FUNCTION_BLOCK FB_MoveZ_Exte
VAR_INPUT
	ref		:AXIS_REF;
	jogF	:BOOL;
	jogB	:BOOL;
	PosLimit			:BOOL;			(*正极限位信号*)
	NegLimit			:BOOL;			(*负极限位信号*)
	electromagnetLimit	:BOOL;
	
	maxDistance			:LREAL;			(*最大行程*)
	Acceleration		:LREAL;
	Deceleration		:LREAL;
	Jerk				:LREAL;
END_VAR
VAR_OUTPUT	
	electromagnet_power :BOOL;
END_VAR
VAR
	MC_Read:MC_ReadStatus;
	MC_ABS:MC_MoveAbsolute;
	MC_REL:MC_MoveRelative;
	MC_Jog:MC_Jog;	
	MC_VELO:MC_MoveVelocity;
	MC_stop:MC_Stop;
	
	step1,step2,step3		:INT;	
	R_TRIG1,R_TRIG2,R_TRIG3	:R_TRIG;
	R_TRIG_done				:R_TRIG;
	ton_NotMoving			:TON;
	ton_Moving				:TON;
	rel_do					:BOOL;
	abs_do					:BOOL;
	jogF_do					:BOOL;
	jogB_do					:BOOL;
	
	velo_do					:BOOL;
	stop_do					:BOOL;
	error					:BOOL;

	MoveAbsolute_Busy		:BOOL;
	MoveVelocity_Busy		:BOOL;
	MoveRelative_Busy		:BOOL;
	jog_EN					:BOOL;
	FB_START_r_trig:		R_TRIG;
	start					:BOOL;
	jog_f_trig				:F_TRIG;
END_VAR
VAR_IN_OUT 
	MoveRelExe					:BOOL;
	MoveAbsExe					:BOOL;
	MoveVelocityExe				:BOOL;//
	Velo						:LREAL;	//mm/s
	TargetRel					:LREAL;//mm
	TargetAbs					:LREAL;//mm
							
	Done						:BOOL;
	NotMovingTimeOut 			:BOOL;
	
END_VAR

(*********************NOT MOVING TIMEOUT***************************)
FB_START_r_trig(CLK:=jogF OR jogB OR MoveRelExe OR MoveAbsExe OR MoveVelocityExe  , Q=> );
IF FB_START_r_trig.Q THEN 
	start:=TRUE;
END_IF
ton_NotMoving(IN:=Ref.Status.NotMoving AND start  , PT:= T#5S, Q=> , ET=> );

Call_FB();
JOG();
MoveAbsolute();
MoveVelocity();
MoveRelative();


(*********************error***************************)
IF ton_NotMoving.Q OR error  THEN	
	start:=FALSE;
	NotMovingTimeOut:=TRUE;	
	error:=FALSE;
	ton_NotMoving(IN:=FALSE);	
	step1:=step2:=step2:=0;	
	MoveRelExe:=FALSE;
	MoveAbsExe:=FALSE;
	MoveVelocityExe:=FALSE;
	TargetAbs:=0;
	TargetRel:=0;
	

	R_TRIG1(CLK:=FALSE);
	R_TRIG2(CLK:=FALSE);
	R_TRIG3(CLK:=FALSE);
END_IF

(*********************move done***************************)
IF MoveAbsolute_Busy OR MoveVelocity_Busy OR  MoveRelative_Busy THEN 
	Done:=FALSE;
	jogF:=FALSE;
	jogB:=FALSE;
END_IF

jog_f_trig(CLK:=jogB OR jogF , Q=> );

R_TRIG_done(CLK:=MC_REL.Done OR MC_ABS.Done OR MC_stop.Done  OR jog_f_trig.Q , Q=> );
IF R_TRIG_done.Q THEN 	
	start:=FALSE;
	R_TRIG_done(CLK:=FALSE);
	NotMovingTimeOut:=FALSE;
	ton_NotMoving(IN:=FALSE);
	step1:=step2:=step2:=0;	
	MoveRelExe:=FALSE;
	MoveAbsExe:=FALSE;
	MoveVelocityExe:=FALSE;
	TargetAbs:=0;
	TargetRel:=0;
	
	Done:=TRUE ;
END_IF

ACTION Call_FB:
MC_Read(
	Axis:=ref , 
	Enable:=TRUE);
MC_REL(
	Axis:=ref , 
	Execute:=rel_do , 
	Distance:=TargetRel , 
	Velocity:=Velo , 
	Acceleration:=Acceleration , 
	Deceleration:=Deceleration , 
	Jerk:=Jerk , 
	BufferMode:= , 
	Options:= , 
	Done=> , 
	Busy=>MoveRelative_Busy , 
	Active=> , 
	CommandAborted=> , 
	Error=> , 
	ErrorID=> );
	IF MC_REL.Busy THEN 
		rel_do:=FALSE;
		MoveRelExe:=FALSE;
	END_IF
MC_ABS(
	Axis:=ref , 
	Execute:=abs_do , 
	Position:=TargetAbs , 
	Velocity:=Velo , 
	Acceleration:=Acceleration , 
	Deceleration:=Deceleration , 
	Jerk:=Jerk , 
	BufferMode:= , 
	Options:= , 
	Done=> , 
	Busy=>MoveAbsolute_Busy , 
	Active=> , 
	CommandAborted=> , 
	Error=> , 
	ErrorID=> );
	IF MC_ABS.Busy THEN 
		abs_do:=FALSE;
		MoveAbsExe:=FALSE;
	END_IF
MC_Jog(
	Axis:=ref , 
	JogForward:=jogF_do , 
	JogBackwards:=jogB_do , 
	Mode:=MC_JOGMODE_CONTINOUS , 
	Position:= , 
	Velocity:=Velo , 
	Acceleration:=Acceleration , 
	Deceleration:=Deceleration , 
	Jerk:=Jerk , 
	Done=> , 
	Busy=> , 
	Active=> , 
	CommandAborted=> , 
	Error=> , 
	ErrorID=> );
MC_VELO(
	Axis:=ref , 
	Execute:=velo_do , 
	Velocity:=Velo , 
	Acceleration:=Acceleration , 
	Deceleration:=Deceleration , 
	Jerk:=Jerk , 
	Direction:= , 
	BufferMode:= MC_Aborting, 
	Options:= , 
	InVelocity=> , 
	Busy=> , 
	Active=> , 
	CommandAborted=> , 
	Error=> , 
	ErrorID=> );
	//IF MC_VELO.Busy THEN 
	//	velo_do:=FALSE;
	//END_IF
MC_stop(
	Axis:=ref , 
	Execute:=stop_do , 
	Deceleration:=Deceleration , 
	Jerk:=Jerk , 
	Options:= , 
	Done=> , 
	Busy=> , 
	Active=> , 
	CommandAborted=> , 
	Error=> , 
	ErrorID=> );
IF MC_stop.Done THEN 
	stop_do:=FALSE;
END_IF
END_ACTION

ACTION JOG:
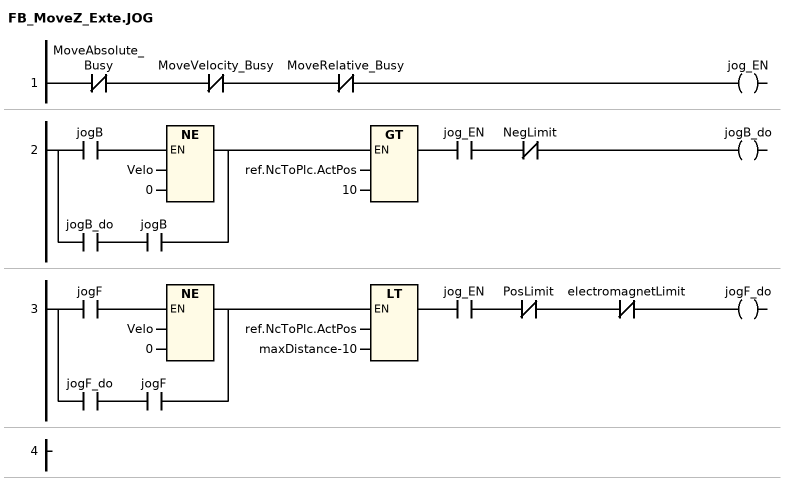
// NETWORK 1
jog_EN := NOT MoveAbsolute_Busy AND NOT MoveVelocity_Busy AND NOT MoveRelative_Busy;

// NETWORK 2
jogB_do := ((jogB AND Velo <> 0 OR jogB_do AND jogB) AND ref.NcToPlc.ActPos > 10) AND jog_EN AND NOT NegLimit;

// NETWORK 3
jogF_do := ((jogF AND Velo <> 0 OR jogF_do AND jogF) AND ref.NcToPlc.ActPos < (maxDistance-10)) AND jog_EN AND NOT PosLimit AND NOT electromagnetLimit;

// NETWORK 4
END_ACTION

ACTION MoveAbsolute:
(****************ABS********************)
R_TRIG2(CLK:=MoveAbsExe AND Ref.Status.NotMoving    , Q=> );

CASE step2 OF 
	0:				
		IF R_TRIG2.Q THEN 
			R_TRIG2(CLK:=FALSE);			
			MoveAbsExe:=FALSE;
			electromagnet_power:=FALSE;
			step2:=1;
		END_IF
	1:	
		IF   Velo<>0 THEN 		
			abs_do:=TRUE;
			step2:=2;
		END_IF
	2:
		IF MC_ABS.Busy THEN 
			abs_do:=FALSE;								
			step2 :=0;
		END_IF	
END_CASE


IF  MoveAbsolute_Busy THEN 
	MoveRelExe:=FALSE;
	MoveVelocityExe:=FALSE;
	electromagnet_power:=FALSE;
END_IF
END_ACTION

ACTION MoveRelative:
(****************Rel********************)
R_TRIG1(CLK:=MoveRelExe AND Ref.Status.NotMoving   , Q=> );
CASE step1 OF 
	0:				
		IF R_TRIG1.Q THEN 
			R_TRIG1(CLK:=FALSE);
			MoveRelExe:=FALSE;
			electromagnet_power:=FALSE;
			step1:=1;
		END_IF
	1:	
		IF TargetRel <>0 AND Velo<>0 THEN 		
			rel_do:=TRUE;
			step1:=2;
		END_IF
	2:
		IF MC_REL.Busy THEN 
			rel_do:=FALSE;								
			step1 :=0;
		END_IF	
END_CASE

IF MoveRelative_Busy THEN 
	MoveAbsExe:=FALSE;
	MoveVelocityExe:=FALSE;
	electromagnet_power:=FALSE;
END_IF
END_ACTION

ACTION MoveVelocity:
(****************当做自动测高********************)
IF electromagnetLimit THEN 
	MoveVelocityExe:=FALSE;
END_IF
R_TRIG3(CLK:=MoveVelocityExe AND Ref.Status.NotMoving AND NOT electromagnetLimit  , Q=> );
CASE step3 OF 
	0:				
		IF R_TRIG3.Q THEN 
			R_TRIG3(CLK:=FALSE);
			MoveVelocityExe:=FALSE;
			velo_do:=FALSE;		
			step3:=1;
		END_IF
	1:	//电磁铁得电
		electromagnet_power:=TRUE;
		IF   Velo<>0 THEN 		
			velo_do:=TRUE;
			step3:=2;
		END_IF
		
	2:	//碰到电磁铁，停止
		IF electromagnetlimit THEN 
			electromagnet_power:=FALSE;
			velo_do:=FALSE;
			stop_do:=TRUE;
			step3 :=0;
		END_IF
END_CASE
MoveVelocity_Busy:=MC_VELO.Busy ;

IF MoveVelocity_Busy THEN 
	MoveRelExe:=FALSE;
	MoveAbsExe:=FALSE;
END_IF
END_ACTION

END_FUNCTION_BLOCK

(* stored: Version 1.1.0.1, ProductVersion 3.1.4024.11
   POU FB_MoveZ_Exte: Id {0b2fc532-d5a8-4eac-8360-efebba4e5c11}, SpecialFunc None
   Action Call_FB: Id {c8dc25fd-fa9e-40a0-b4e1-7f0be54fa570}
   Action JOG: Id {9fa182ac-93ed-4c4c-a649-e44075daf6ca}
   Action MoveAbsolute: Id {9bfbadb9-9d7d-41ed-a9c2-ee2c006bfafb}
   Action MoveRelative: Id {39042831-1f1d-4371-81e1-99bae8284408}
   Action MoveVelocity: Id {888180fb-a6be-4e8d-b014-2b51b528a886} *)
